TYPE UnitIndexerMaster EXTENDS UnitBase :
	//6
STRUCT
	guidUpstream : DWORD;//16-17
	slaveLinkageStatus : DWORD;//18-19 , 32 slave linkage possible
	//
	reserved : ARRAY[1..12] OF WORD; // 20-31
	// 64bytes , 32 word occupation here
	
	//isSyncEngaged : BOOL; //32
	//matIsValidStatus : DWORD;
	//matSyncDone : DWORD;
	//slaveWorkingSignal : DWORD;
	//syncWord : WORD; //sync is working , sync first time
	
END_STRUCT
END_TYPE

(* stored: Version 1.1.0.1, ProductVersion 3.1.4022.10
   DUT UnitIndexerMaster: Id {4e22941b-cab4-4ec7-873b-1c5ab67c30f9} *)
